// TIA Portal V17 export
// export: Created 2022-07-20T07:02:39.8574443Z, ExportSetting WithDefaults, DisplayName Totally Integrated Automation Portal, DisplayVersion V17, DisplayName TIA Portal Openness, DisplayVersion V17, DisplayName TIA Portal Version Control Interface, DisplayVersion V17, DisplayName SINAMICS Startdrive Advanced, DisplayVersion V17, DisplayName SINAMICS Startdrive G130, G150, S120, S150, SINAMICS MV, S210, DisplayVersion V17, DisplayName SINAMICS Startdrive G110M, G120, G120C, G120D, G120P, G115D, DisplayVersion V17, DisplayName STEP 7 Professional, DisplayVersion V17, DisplayName STEP 7 Safety, DisplayVersion V17, DisplayName WinCC Advanced, DisplayVersion V17
VAR_GLOBAL   // PLC tag table "LCamHdl_ProfileConstants"
END_VAR
VAR_GLOBAL CONSTANT   // user constants
   LCAMHDL_PROFILE_EMPTY : DInt := 0;
   LCAMHDL_PROFILE_POINT : DInt := 1;
   LCAMHDL_PROFILE_DWELL : DInt := 2;
   LCAMHDL_PROFILE_CONST_VELO : DInt := 3;
   LCAMHDL_PROFILE_POLY_3 : DInt := 4;
   LCAMHDL_PROFILE_POLY_5 : DInt := 5;
   LCAMHDL_PROFILE_POLY_7 : DInt := 6;
   LCAMHDL_PROFILE_D_D_PARABOLA : DInt := 7;
   LCAMHDL_PROFILE_C_C_PARABOLA : DInt := 8;
   LCAMHDL_PROFILE_D_D_BASIC_SINE : DInt := 9;
   LCAMHDL_PROFILE_D_D_INCLINED_SINE : DInt := 10;
   LCAMHDL_PROFILE_D_D_MOD_ACCEL_TRAPEZOID : DInt := 11;
   LCAMHDL_PROFILE_D_D_MOD_SINE : DInt := 12;
   LCAMHDL_PROFILE_C_C_MOD_SINE : DInt := 13;
   LCAMHDL_PROFILE_R_R_MOD_VELO_TRAPEZOID : DInt := 14;
   LCAMHDL_PROFILE_R_R_BASIC_SINE : DInt := 15;
   LCAMHDL_PROFILE_D_C_MOD_SINE : DInt := 16;
   LCAMHDL_PROFILE_C_D_MOD_SINE : DInt := 17;
   LCAMHDL_PROFILE_D_R_MOD_ACCEL_TRAPEZOID : DInt := 18;
   LCAMHDL_PROFILE_R_D_MOD_ACCEL_TRAPEZOID : DInt := 19;
   LCAMHDL_PROFILE_D_R_HARMONIC_COMBINATION : DInt := 20;
   LCAMHDL_PROFILE_R_D_HARMONIC_COMBINATION : DInt := 21;
   LCAMHDL_PROFILE_C_R_HARMONIC_COMBINATION : DInt := 22;
   LCAMHDL_PROFILE_R_C_HARMONIC_COMBINATION : DInt := 23;
   LCAMHDL_PROFILE_POLY_4 : DInt := 30;
   LCAMHDL_PROFILE_POLY_6 : DInt := 35;
   LCAMHDL_ADD_PROFILE_POLY : DInt := 44;
   LCAMHDL_ADD_PROFILE_POLY_TRIGONOMETRIC : DInt := 45;
   LCAMHDL_ADD_PROFILE_SINE : DInt := 51;
   LCAMHDL_ADD_PROFILE_INCLINED_SINE : DInt := 52;
   LCAMHDL_ADD_PROFILE_INVERSE_SINE : DInt := 55;
   LCAMHDL_ADD_PROFILE_D_R_DOUBLE_HARMONIC : DInt := 60;
   LCAMHDL_ADD_PROFILE_R_D_DOUBLE_HARMONIC : DInt := 61;
END_VAR
